PROGRAM switch
VAR
	fbRecGeneric		: 	FB_Rec_Generic;
END_VAR
VAR_INPUT
	sensorID			: DWORD;
END_VAR
VAR_OUTPUT
	switchNR			: INT;
END_VAR

fbRecGeneric(str_KL6581 := GVL_EnOcean.stKL6581, byNode := 0, dw_ID := sensorID);

IF fbRecGeneric.bReceive = FALSE THEN
	IF fbRecGeneric.ar_Value[3] = 16 THEN
		switchNR := 1;
	ELSIF fbRecGeneric.ar_Value[3] = 80 THEN
		switchNR := 2;
	ELSIF fbRecGeneric.ar_Value[3] = 96 THEN
		switchNR := 3;
	ELSIF fbRecGeneric.ar_Value[3] = 112 THEN
		switchNR := 4;
	ELSE 
		switchNR := 0;
	END_IF
END_IF

END_PROGRAM

(* stored: Version 1.1.0.1, ProductVersion 3.1.4022.17
   POU switch: Id {98e622f1-635d-4cae-80de-7cc30f8c4b9a}, SpecialFunc None *)
